FUNCTION_BLOCK SS5b_Raiser_n_Flipper (* Basic FB with empty ECC *)
  (* Standard: 61499-2 *)
  (* Version 1.0, 2024-10-03, DEVIASH *)
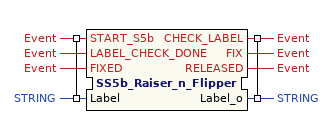
  EVENT_INPUT
    START_S5b WITH Label;
    LABEL_CHECK_DONE;
    FIXED;
  END_EVENT
  EVENT_OUTPUT
    CHECK_LABEL WITH Label_o;
    FIX;
    RELEASED;
  END_EVENT
  VAR_INPUT
    Label : STRING;
  END_VAR
  VAR_OUTPUT
    Label_o : STRING;
  END_VAR
  VAR
    iCount : SINT;
  END_VAR
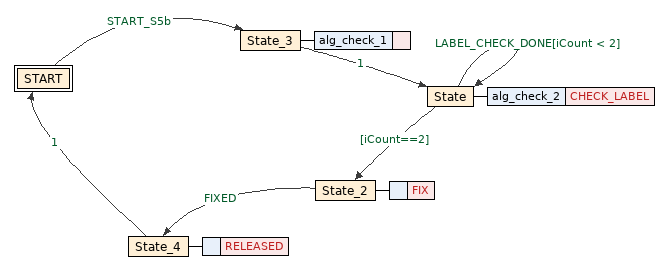
  EC_STATES
    START; (* Initial State *)
    State : alg_check_2 -> CHECK_LABEL;
    State_2 : -> FIX;
    State_3 : alg_check_1;
    State_4 : -> RELEASED;
  END_STATES
  EC_TRANSITIONS
    START TO State_3 := START_S5b;
    State_3 TO State := 1;
    State TO State := LABEL_CHECK_DONE[iCount < 2];
    State TO State_2 := [iCount==2];
    State_2 TO State_4 := FIXED;
    State_4 TO START := 1;
  END_TRANSITIONS
  ALGORITHM alg_check_1 IN ST:
iCount = 0;
  END_ALGORITHM
  ALGORITHM alg_check_2 IN ST:
iCount = iCount + 1;
  END_ALGORITHM
END_FUNCTION_BLOCK
